PROGRAM PRG_AtEntry02
VAR
	intnFBSensor : FB_Sensors;
	FEdge : F_TRIG;
END_VAR

intnFBSensor (
	iSensor := At_Entry_2,
	iTimeToActuateSensor := 0,
);

FEdge (
	CLK := intnFBSensor.outSensorON,
);

END_PROGRAM

(* stored: Version 1.1.0.1
   POU PRG_AtEntry02: Id {4e5493cd-88f3-4e14-b9fc-27d34b252294}, SpecialFunc None *)
